TYPE Port_Map :
STRUCT
	JBOX_PORT : STRING(5);
	TESTER_PORT : STRING(5);
END_STRUCT
END_TYPE

(* stored: Version 1.1.0.1, ProductVersion 3.1.4024.10
   DUT Port_Map: Id {ea999e49-017a-4c9f-9c84-f9ad6b83ea86} *)
